PROGRAM MAIN
VAR
	AXIS1:axis_ref;
	POWER1:mc_power;
	power_do: BOOL;

	move_abs: MC_MoveAbsolute;
	abs_do: BOOL;
	position: LREAL;
	vel: LREAL;
END_VAR

POWER1(
	Axis:= AXIS1, 
	Enable:= power_do, 
	Enable_Positive:= TRUE, 
	Enable_Negative:= TRUE, 
	Override:= , 
	BufferMode:= , 
	Options:= , 
	Status=> , 
	Busy=> , 
	Active=> , 
	Error=> , 
	ErrorID=> );
	
move_abs(
	Axis:= AXIS1, 
	Execute:= abs_do, 
	Position:= position, 
	Velocity:= vel, 
	Acceleration:= , 
	Deceleration:= , 
	Jerk:= , 
	BufferMode:= , 
	Options:= , 
	Done=> , 
	Busy=> , 
	Active=> , 
	CommandAborted=> , 
	Error=> , 
	ErrorID=> );

END_PROGRAM

(* stored: Version 1.1.0.1, ProductVersion 3.1.4024.5
   POU MAIN: Id {c77aa319-5c1d-4123-b1e2-660c87d39da9}, SpecialFunc None *)
